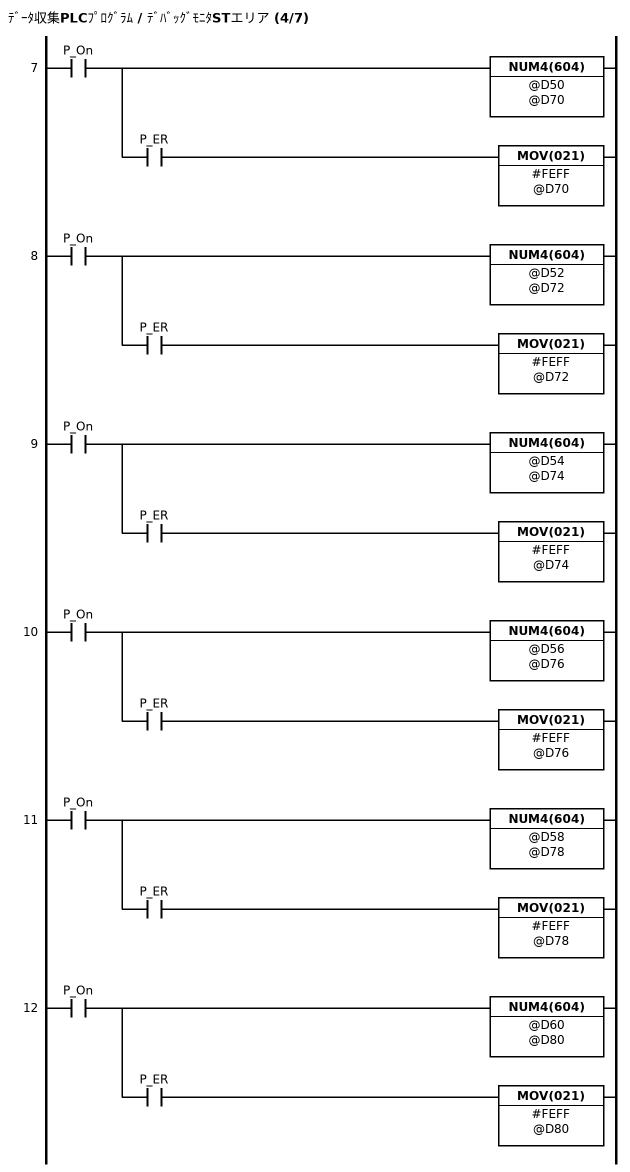
; [picture p48: ﾃﾞｰﾀ収集PLCﾌﾟﾛｸﾞﾗﾑ / ﾃﾞﾊﾞｯｸﾞﾓﾆﾀSTエリア, rungs 7-12]
; rung 7
LD P_On
NUM4(604) @D50 @D70
AND P_ER
MOV(021) #FEFF @D70
; rung 8
LD P_On
NUM4(604) @D52 @D72
AND P_ER
MOV(021) #FEFF @D72
; rung 9
LD P_On
NUM4(604) @D54 @D74
AND P_ER
MOV(021) #FEFF @D74
; rung 10
LD P_On
NUM4(604) @D56 @D76
AND P_ER
MOV(021) #FEFF @D76
; rung 11
LD P_On
NUM4(604) @D58 @D78
AND P_ER
MOV(021) #FEFF @D78
; rung 12
LD P_On
NUM4(604) @D60 @D80
AND P_ER
MOV(021) #FEFF @D80

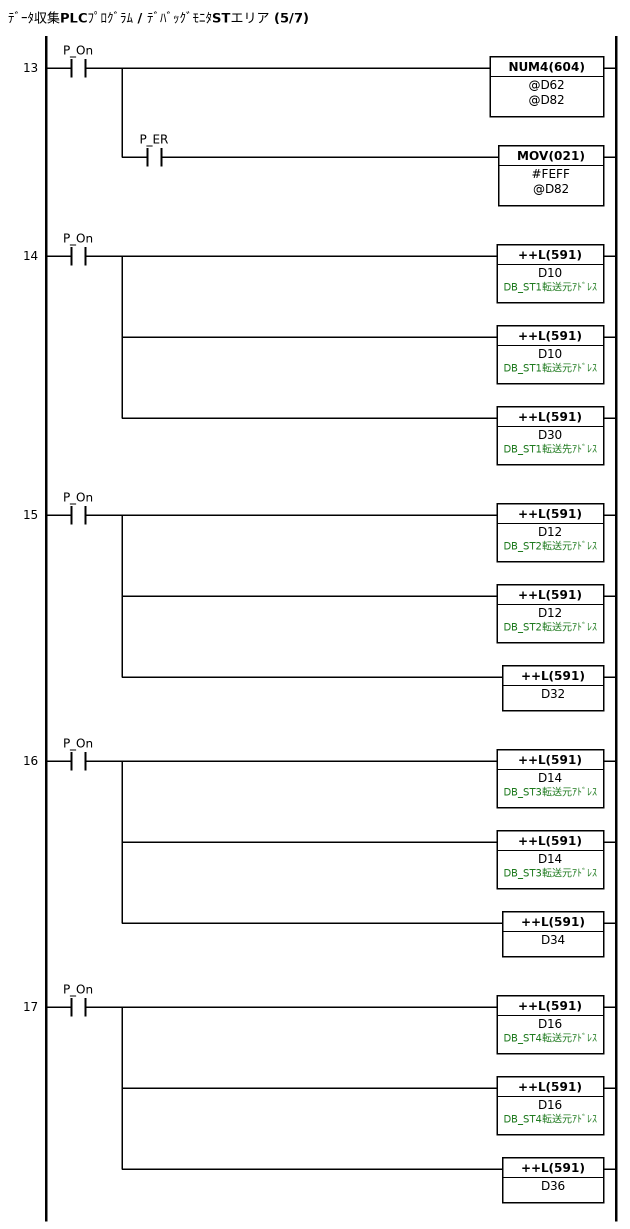
; rung 13
LD P_On
NUM4(604) @D62 @D82
AND P_ER
MOV(021) #FEFF @D82
; rung 14
LD P_On
++L(591) D10  ; DB_ST1転送元ｱﾄﾞﾚｽ
++L(591) D10  ; DB_ST1転送元ｱﾄﾞﾚｽ
++L(591) D30  ; DB_ST1転送先ｱﾄﾞﾚｽ
; rung 15
LD P_On
++L(591) D12  ; DB_ST2転送元ｱﾄﾞﾚｽ
++L(591) D12  ; DB_ST2転送元ｱﾄﾞﾚｽ
++L(591) D32
; rung 16
LD P_On
++L(591) D14  ; DB_ST3転送元ｱﾄﾞﾚｽ
++L(591) D14  ; DB_ST3転送元ｱﾄﾞﾚｽ
++L(591) D34
; rung 17
LD P_On
++L(591) D16  ; DB_ST4転送元ｱﾄﾞﾚｽ
++L(591) D16  ; DB_ST4転送元ｱﾄﾞﾚｽ
++L(591) D36

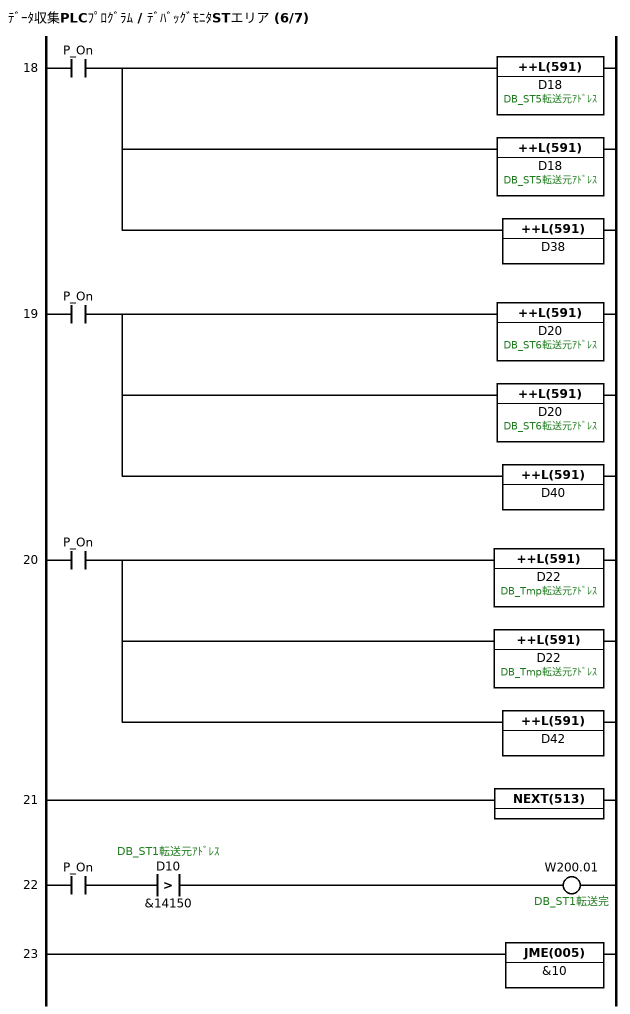
; rung 18
LD P_On
++L(591) D18  ; DB_ST5転送元ｱﾄﾞﾚｽ
++L(591) D18  ; DB_ST5転送元ｱﾄﾞﾚｽ
++L(591) D38
; rung 19
LD P_On
++L(591) D20  ; DB_ST6転送元ｱﾄﾞﾚｽ
++L(591) D20  ; DB_ST6転送元ｱﾄﾞﾚｽ
++L(591) D40
; rung 20
LD P_On
++L(591) D22  ; DB_Tmp転送元ｱﾄﾞﾚｽ
++L(591) D22  ; DB_Tmp転送元ｱﾄﾞﾚｽ
++L(591) D42
; rung 21
NEXT(513)
; rung 22
LD P_On
AND>L(321) D10 &14150  ; DB_ST1転送元ｱﾄﾞﾚｽ
OUT W200.01  ; DB_ST1転送完
; rung 23
JME(005) &10

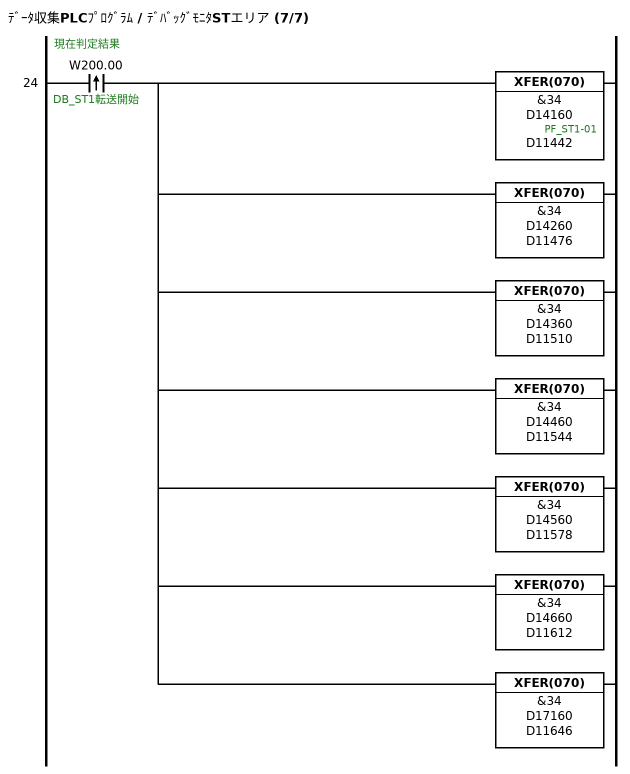
; rung 24: 現在判定結果
@LD W200.00  ; DB_ST1転送開始
XFER(070) &34 D14160 D11442  ; PF_ST1-01
XFER(070) &34 D14260 D11476
XFER(070) &34 D14360 D11510
XFER(070) &34 D14460 D11544
XFER(070) &34 D14560 D11578
XFER(070) &34 D14660 D11612
XFER(070) &34 D17160 D11646

### Section END
; rung 0
END(001)